(*********************************** G.D S.p.A. - Technical Department ***********************************
============= PROGRAM INFO ============
FOLDER:             TBD
MACHINES INVOLVED:  TBD 

============= DESCRIPTION =============
csp machine declaration

============= REVISIONS ===============
Date		Version	 	Author      	Description             
----------	-------		------------  	--------------------------------------------
2019/04/05 	0000.00	 	M.Grasso		Creation of the PRG

**********************************************************************************************************)
(*$R process_ref := prc; $*)
PROGRAM csp_case_fc_os_upper_sensors
VAR
	
	prc:											process;
	prc_path:										STRING;
	
	flap_chksect:									check_section;
	flap_inchoerence_chksect:						check_section;
	bad_count:										INT;
	consecutive_reject_aem:							message;
	check_request_rtrig:							R_TRIG;
	check_request:									BOOL;
	
	consecutive_blocked_aem:						message;
	blocked_latch:									BOOL;
	consecutive_blocked_count:						INT;
	max_OS_upper_sensor_fail_nvr:					INT := 2; (*$P min:=2; max:=30; $*)
	
END_VAR
VAR_INPUT
	flap_di:										digital_input;
END_VAR

_read_var_input();

_object_manager();

IF NOT objects_running()
THEN
	RETURN;	
END_IF

_read_process_image();

_mode_manager();

_set_runtime_properties();

(********************************* BODY *********************************)
check_section_message_disable(flap_chksect);

check_section_set_check_window_phases_value(
    begin_phase         :=  csp_case_flapControl.Flap_check_begin_phase,
    end_phase           :=  csp_case_flapControl.Flap_check_end_phase,
    conversion_THIS     :=  flap_chksect);	
	
IF csp_case_main_services.dry_cycle_mode
	OR csp_main_motorization.empty_command
THEN
	check_section_disable(flap_chksect);
ELSE
	check_section_enable(flap_chksect);
END_IF

check_request_rtrig(CLK := csp_case_feed_virtualMaster.follower_check_request);
check_request := check_request_rtrig.Q;

(* TRACKS IF PE WAS BAD DURING REJECT *)
IF phase_window_falling_edge(csp_case_transport_virtualMaster.major_flap_phwin)
	OR
	(
		//csp_case_feed_virtualMaster.follower_check_request
		check_request
		AND csp_case_transport.flap_control_axes_standstill
		AND csp_case_transport.Followers_Extended
		AND csp_case_transport.Spreaders_Extended
	)
	AND NOT digital_input_is_active(flap_di)
THEN
	bad_count :=  bad_count + 1;
END_IF

IF csp_case_transport_virtualMaster.PE_check
	OR machine_is_stopped(csp.mch)
	OR machine_is_stop_emergency_active(csp.mch)
	OR csp_main_motorization.empty_command
THEN
	bad_count := 0;
	process_message_reset(consecutive_reject_aem);
END_IF

IF 	bad_count >= max_OS_upper_sensor_fail_nvr
	AND NOT csp_main_motorization.empty_command
THEN
	process_message_set(1, 1, 1, consecutive_reject_aem);
END_IF


(* TO MONITOR CONSECUTIVE BLOCKED PE *)
IF 	phase_window_position_is_in_window(csp_case_transport_virtualMaster.axis.actual_position, csp_case_flapControl.consecutive_blocked_phwin)
	AND digital_input_is_active(flap_di)
THEN
	blocked_latch := TRUE;
END_IF

IF 	blocked_latch
	AND phase_window_falling_edge(csp_case_flapControl.consecutive_blocked_phwin)
THEN
	consecutive_blocked_count := consecutive_blocked_count + 1;
END_IF

(* CLEARS COUNT IF EVER NOT BLOCKED *)
IF 	NOT digital_input_is_active(flap_di)
THEN
	blocked_latch := FALSE;
	consecutive_blocked_count := 0;
END_IF

(* TURNS ON MESSAGE IF CONSECUTIVE *)
IF 	consecutive_blocked_count >= max_OS_upper_sensor_fail_nvr
THEN
	process_message_set(1, 1, 1, consecutive_blocked_aem);
END_IF

IF 	machine_is_stopped(csp.mch)
	OR machine_is_stop_emergency_active(csp.mch)
THEN
	process_message_reset(consecutive_blocked_aem);
	blocked_latch := FALSE;
	consecutive_blocked_count := 0;
END_IF


(************************************************************************)

_handle_messages();

_write_output();

ACTION _handle_messages:
;
END_ACTION

ACTION _handle_process_test:
;
END_ACTION

ACTION _mode_manager:
IF process_mode_req_is_pending(prc)
THEN
    process_apply_mode_req_first_step(prc);
    CASE process_get_mode(prc) OF
        MODE_TO_ABSENT:
			;
        MODE_TO_INACTIVE:
			;
        MODE_TO_TEST:
			;
        MODE_TO_OPERATIONAL:
			;
    END_CASE
    process_apply_mode_req_second_step(prc);
END_IF
END_ACTION

ACTION _object_manager:
IF objects_initialization()
THEN
	sub_process_init(
		object_name					:= 'csp_case_fc_os_upper_sensors.prc', 
		process						:= csp_case_fc_os_upper.prc, 
		CONVERSION_this				:= prc);
		
	prc_path 						:= process_get_path(prc);
	
	(* INPUTS *)
	digital_input_init(
		object_name					:= CONCAT(prc_path, '_flap_di'), 
		polarity_direct				:= TRUE, 
		process						:= prc, 
		CONVERSION_this				:= flap_di);
	
(* CHECK SECTION FOR THE OPERATOR SIDE UPPER FLAP SETS SHIFT REGISTER AND PE FAILURE LOGIC *)	
	check_section_window_mode_init(
        object_name:= CONCAT(prc_path, '_flap_chksect'),
        check_enable:= TRUE,
        event_to_check:= CHECK_SECTION_EVENT_INPUT_ON,
        execution_mode:=  CHECK_SECTION_EXECUTION_WHEN_EVENT_OCCURRED,
        diagnostic_enable:= FALSE,
        status_bits_to_be_true:= common_global_variables.NONE,//ITEM_CASE_FEED,//AMR 9/1/2021
        status_bits_to_be_false:= common_global_variables.NONE,
        _step_status_conditioning_execution:= FALSE,
        status_bits_to_set:= common_global_variables.NONE,//ITEM_HAS_OS_UPPER_FLAP,//AMR 9/1/2021
        status_bits_to_reset:= common_global_variables.NONE,
        reject_bit_to_set:= 0,
        _step:= 25,
        first_step_to_write_offset:= 0,
        number_of_steps_to_write:= 1,
        begin_phase:= csp_case_flapControl.Flap_check_begin_phase,
        end_phase:= csp_case_flapControl.Flap_check_end_phase,
        max_consecutive_failed_checks:= 3,
        max_failed_checks_percentage:= 100,
        products_for_failed_checks_percentage:= 10,
        shift_register:= csp_case_main_statistics.sr ,
        process:= prc,
        CONVERSION_this:= flap_chksect );

	check_section_add_di_input(
		di_input := flap_di,
		CONVERSION_this:= flap_chksect);
	
	message_configure(
        individual_reset                    := FALSE,
        machine_reaction                    := MACHINE_REACTION_STOP_IN_PHASE_ONE,
        typology                            := MESSAGE_TYPOLOGY_ABNORMAL,
        CONVERSION_this                     := flap_chksect.too_many_failed_checks_aem.message );	
		
		
 	check_section_window_mode_init(
		object_name:= CONCAT(prc_path, '_flap_inchoerence_chksect'),
		check_enable:= TRUE, 
		event_to_check:= CHECK_SECTION_EVENT_INPUT_ALWAYS_ON, 
		execution_mode:= CHECK_SECTION_EXECUTION_WHEN_EVENT_OCCURRED, 
		diagnostic_enable:= FALSE, 
		status_bits_to_be_true:= 0, 
		status_bits_to_be_false:= 0, 
		_step_status_conditioning_execution:= FALSE, 
		status_bits_to_set:= 0, 
		status_bits_to_reset:= 0, 
		reject_bit_to_set:= 0, 
		_step:= 25, 
		first_step_to_write_offset:= 0, 
		number_of_steps_to_write:= 1, 
		begin_phase:= 175, 
		end_phase:= 180, 
		max_consecutive_failed_checks:= 3, 
		max_failed_checks_percentage:= 100, 
		products_for_failed_checks_percentage:= 100, 
		shift_register:= csp_case_main_statistics.sr , 
		process:= prc, 
		CONVERSION_this:= flap_inchoerence_chksect );

	check_section_add_di_input(
		di_input := flap_di,
		CONVERSION_this:= flap_inchoerence_chksect);

	message_configure(
        individual_reset                    := FALSE,
        machine_reaction                    := MACHINE_REACTION_STOP_IN_PHASE_ONE,
        typology                            := MESSAGE_TYPOLOGY_ABNORMAL,
        CONVERSION_this                     := flap_inchoerence_chksect.too_many_failed_checks_aem.message );	
		
	process_message_init(
		object_name:= CONCAT(prc_path, '_consecutive_reject_aem'), 
		behaviour:= MESSAGE_BEHAVIOUR_STATE, 
		reset_timeout:= 0, 
		disableable:= FALSE, 
		individual_reset:= FALSE, 
		machine_reaction:= MACHINE_REACTION_STOP_IN_PHASE_ONE, 
		typology:= MESSAGE_TYPOLOGY_ABNORMAL, 
		process:= prc, 
		CONVERSION_this:= consecutive_reject_aem);
		
	process_message_init(
		object_name:= CONCAT(prc_path, '_consecutive_blocked_aem'), 
		behaviour:= MESSAGE_BEHAVIOUR_STATE, 
		reset_timeout:= 0, 
		disableable:= FALSE, 
		individual_reset:= FALSE, 
		machine_reaction:= MACHINE_REACTION_STOP_IN_PHASE_ONE, 
		typology:= MESSAGE_TYPOLOGY_ABNORMAL, 
		process:= prc, 
		CONVERSION_this:= consecutive_blocked_aem);
		
END_IF

IF objects_running()
THEN
	process_cycle(prc);
	
END_IF
END_ACTION

ACTION _read_process_image:
;
END_ACTION

ACTION _read_var_input:
;
END_ACTION

ACTION _set_runtime_properties:
;
END_ACTION

ACTION _write_output:
;
END_ACTION

END_PROGRAM

(* stored: Version 1.1.0.1, ProductVersion 3.1.4024.3
   POU csp_case_fc_os_upper_sensors: Id {64b0a09b-1866-49ef-add5-41245d359115}, SpecialFunc None
   Action _handle_messages: Id {caedea72-b7ee-4668-9660-6fd698629cdc}
   Action _handle_process_test: Id {cf803617-eaa6-4be8-90c5-f6c4e38ff064}
   Action _mode_manager: Id {51a99b7d-3fac-4668-88bf-eaf12920c503}
   Action _object_manager: Id {02b09c87-4f7d-48d7-bdfe-adc0677271de}
   Action _read_process_image: Id {eaf7a2e4-d93d-417a-b97f-af0fb36a0041}
   Action _read_var_input: Id {31aca0a8-9e3e-4fd6-af08-d42543ed1a87}
   Action _set_runtime_properties: Id {61e8e8d3-002a-4ba4-8314-0120275c4378}
   Action _write_output: Id {f44a4638-7fbc-4b41-9bef-f28d203be274} *)
